PROGRAM MAIN
VAR
END_VAR

END_PROGRAM

(* stored: Version 1.1.0.1
   POU MAIN: Id {88148cc8-699f-4d2c-9a91-ef92502d4b11} *)
